{attribute 'qualified_only'}
{attribute 'strict'}
TYPE Command :
(
    Off := 0,
    On
);
END_TYPE

(* stored: Version 1.1.0.1, ProductVersion 3.1.4024.4
   DUT Command: Id {c3a73ade-78fa-488c-9caf-5ad1502b78a6} *)
